FUNCTION_BLOCK UnitTestRunner IMPLEMENTS IRunner
VAR_INPUT
END_VAR
VAR_OUTPUT
END_VAR
VAR
    testSuites: ARRAY [0..10] OF ITestSuite;
END_VAR

PROPERTY numberOfTestSuites : UINT
GET
VAR
    i: INT;
END_VAR
numberOfTestSuites := 0;
FOR i:=0 TO 10 DO
    IF THIS^.testSuites[i] <> 0 THEN
        numberOfTestSuites := numberOfTestSuites + 1;
    ELSE
        EXIT;
	END_IF
END_FOR
END_GET
END_PROPERTY

METHOD registerTestSuite
VAR_INPUT
    testSuite: ITestSuite;
END_VAR
VAR
    i: INT;
END_VAR
FOR i:=0 TO 10 DO
    IF THIS^.testSuites[i] = testSuite THEN
        EXIT;
	END_IF
    IF THIS^.testSuites[i] = 0 THEN
        THIS^.testSuites[i] := testSuite;
        EXIT;
	END_IF
END_FOR
END_METHOD

METHOD runAllTests
VAR
    i: INT;
END_VAR
FOR i:=0 TO 10 DO
    IF testSuites[i] = 0 THEN
        EXIT;
	END_IF
    testSuites[i].runAllTests();
END_FOR
END_METHOD

END_FUNCTION_BLOCK

(* stored: Version 1.1.0.1, ProductVersion 3.1.4022.12
   POU UnitTestRunner: Id {3037e080-9321-446b-b115-077ca09a8178}, SpecialFunc None
   Property numberOfTestSuites: Id {69763f75-f9ae-48ad-b38b-91669c6f8622}
   Get Get: Id {dbe5fc45-3eb6-4b00-9d8b-b2fe05ff8daa}
   Method registerTestSuite: Id {9a359b67-3d70-4fc5-8498-38bc8aec6f8b}
   Method runAllTests: Id {3d38c77b-c7eb-45cc-82bd-431fcedeb6a9} *)
